PROGRAM To_Do_List
VAR
END_VAR

(*

Create Wireless Enable
OR Joystick buttons

Add Joystick Estop to PLC estop

Calibrate Joystick















*)

END_PROGRAM

(* stored: Version 1.1.0.1, ProductVersion 3.1.4022.3
   POU To_Do_List: Id {6aec0084-8702-45f9-8721-b3ccb8499ec5}, SpecialFunc None *)
